// TIA Portal V18 export
// export: Created 2025-12-01T12:38:33.7594151Z, ExportSetting None, DisplayName Totally Integrated Automation Portal, DisplayVersion V18 Update 5, DisplayName TIA Portal Openness, DisplayVersion V18 Update 5, DisplayName TIA Portal Teamcenter Gateway, DisplayVersion V18, DisplayName TIA Portal Version Control Interface, DisplayVersion V18, DisplayName STEP 7 Professional, DisplayVersion V18 Update 5, DisplayName STEP 7 Safety, DisplayVersion V18, DisplayName WinCC Professional, DisplayVersion V18 Update 5
FUNCTION "ST10Cyl_interface41-50" : Void   // FC1024, LAD
{ S7_Optimized_Access := 'FALSE' }
// stored: AutoNumber false, SetENOAutomatically false
   VAR_INPUT
      AlwaysON : Bool;
      E_stop : Bool;
   END_VAR
   VAR_TEMP
      tTest : Bool;
   END_VAR
BEGIN

REGION Network 1 (SCL): Cylinder 41-50 IO Interface (SCL)
   //Cylinder41 IO  K-reserveLifting3LiftingCylinder
   //Input
   "ST10Cylinder".Cy[41].In.WorkPositionSensor := "iK-reserveLifting3LiftingCylinderInWP";
   "ST10Cylinder".Cy[41].In.HomePositionSensor := "iK-reserveLifting3LiftingCylinderInHP";
   //Output
   "oK-reserveLifting3LiftingCylinderToWP" := "ST10Cylinder".Cy[41].Out.GoWorkPosition;
   "oK-reserveLifting3LiftingCylinderToHP" := "ST10Cylinder".Cy[41].Out.GoHomePosition;

   //Cylinder42 IO  K-reserveLifting3PalletLocationCylinder
   //Input
   "ST10Cylinder".Cy[42].In.WorkPositionSensor := "iK-reserveLifting3PalletLocationCylinderInWP";
   "ST10Cylinder".Cy[42].In.HomePositionSensor := "iK-reserveLifting3PalletLocationCylinderInHP";
   //Output
   "oK-reserveLifting3PalletLocationCylinderToWP" := "ST10Cylinder".Cy[42].Out.GoWorkPosition;
   "oK-reserveLifting3PalletLocationCylinderToHP" := "ST10Cylinder".Cy[42].Out.GoHomePosition;

   //Cylinder43 IO  K-reserveLoadingStopperCylinder1
   //Input
   "ST10Cylinder".Cy[43].In.WorkPositionSensor := "oK-reserveLoadingStopperCylinder1_ToWP";
   "ST10Cylinder".Cy[43].In.HomePositionSensor := "oK-reserveLoadingStopperCylinder1_ToHP";
   //Output
   "oK-reserveLoadingStopperCylinder1_ToWP" := "ST10Cylinder".Cy[43].Out.GoWorkPosition;
   "oK-reserveLoadingStopperCylinder1_ToHP" := "ST10Cylinder".Cy[43].Out.GoHomePosition;

   //Cylinder44 IO  K-reserveLoadingStopperCylinder2
   //Input
   "ST10Cylinder".Cy[44].In.WorkPositionSensor := "oK-reserveLoadingStopperCylinder2_ToWP";
   "ST10Cylinder".Cy[44].In.HomePositionSensor := "oK-reserveLoadingStopperCylinder2_ToHP";
   //Output
   "oK-reserveLoadingStopperCylinder2_ToWP" := "ST10Cylinder".Cy[44].Out.GoWorkPosition;
   "oK-reserveLoadingStopperCylinder2_ToHP" := "ST10Cylinder".Cy[44].Out.GoHomePosition;

   //Cylinder45 IO  K-reserveLoadingStopperCylinder3
   //Input
   "ST10Cylinder".Cy[45].In.WorkPositionSensor := "oK-reserveLoadingStopperCylinder3_ToWP";
   "ST10Cylinder".Cy[45].In.HomePositionSensor := "oK-reserveLoadingStopperCylinder3_ToHP";
   //Output
   "oK-reserveLoadingStopperCylinder3_ToWP" := "ST10Cylinder".Cy[45].Out.GoWorkPosition;
   "oK-reserveLoadingStopperCylinder3_ToHP" := "ST10Cylinder".Cy[45].Out.GoHomePosition;

   //Cylinder46 K-reserveLoadingStopperCylinder4
   //Input
   "ST10Cylinder".Cy[46].In.WorkPositionSensor := "oK-reserveLoadingStopperCylinder4_ToWP";
   "ST10Cylinder".Cy[46].In.HomePositionSensor := "oK-reserveLoadingStopperCylinder4_ToHP";
   //Output
   "oK-reserveLoadingStopperCylinder4_ToWP" := "ST10Cylinder".Cy[46].Out.GoWorkPosition;
   "oK-reserveLoadingStopperCylinder4_ToHP" := "ST10Cylinder".Cy[46].Out.GoHomePosition;

   //Cylinder47 K-reserveTakeStopperCylinder1
   //Input
   "ST10Cylinder".Cy[47].In.WorkPositionSensor := "oK-reserveTakeStopperCylinder1_ToWP";
   "ST10Cylinder".Cy[47].In.HomePositionSensor := "oK-reserveTakeStopperCylinder1_ToHP";
   //Output
   "oK-reserveTakeStopperCylinder1_ToWP" := "ST10Cylinder".Cy[47].Out.GoWorkPosition;
   "oK-reserveTakeStopperCylinder1_ToHP" := "ST10Cylinder".Cy[47].Out.GoHomePosition;

   //Cylinder48 K-reserveTakeStopperCylinder2
   //Input
   "ST10Cylinder".Cy[48].In.WorkPositionSensor := "oK-reserveTakeStopperCylinder2_ToWP";
   "ST10Cylinder".Cy[48].In.HomePositionSensor := "oK-reserveTakeStopperCylinder2_ToHP";
   //Output
   "oK-reserveTakeStopperCylinder2_ToWP" := "ST10Cylinder".Cy[48].Out.GoWorkPosition;
   "oK-reserveTakeStopperCylinder2_ToHP" := "ST10Cylinder".Cy[48].Out.GoHomePosition;

   //Cylinder49 K-reserveTakeStopperCylinder3
   //Input
   "ST10Cylinder".Cy[49].In.WorkPositionSensor := "oK-reserveTakeStopperCylinder3_ToWP";
   "ST10Cylinder".Cy[49].In.HomePositionSensor := "oK-reserveTakeStopperCylinder3_ToHP";
   //Output
   "oK-reserveTakeStopperCylinder3_ToWP" := "ST10Cylinder".Cy[49].Out.GoWorkPosition;
   "oK-reserveTakeStopperCylinder3_ToHP" := "ST10Cylinder".Cy[49].Out.GoHomePosition;

   (*
   //Cylinder50 K-reserveLoadingStopperCylinder4_2
   // //Input
   "ST10Cylinder".Cy[50].In.WorkPositionSensor := "oK-reserveLoadingStopperCylinder4_2";
   "ST10Cylinder".Cy[50].In.HomePositionSensor := NOT "oK-reserveLoadingStopperCylinder4_2";
   // //Output
   "oK-reserveLoadingStopperCylinder4_2" := "ST10Cylinder".Cy[50].Out.GoWorkPosition;
   // "Feeding washer  lift Cylinder ToHP" := "ST10Cylinder".Cy[50].Out.GoHomePosition;
   *)
END_REGION

REGION Network 2: CY41 interface K-reserveLifting3LiftingCylinder
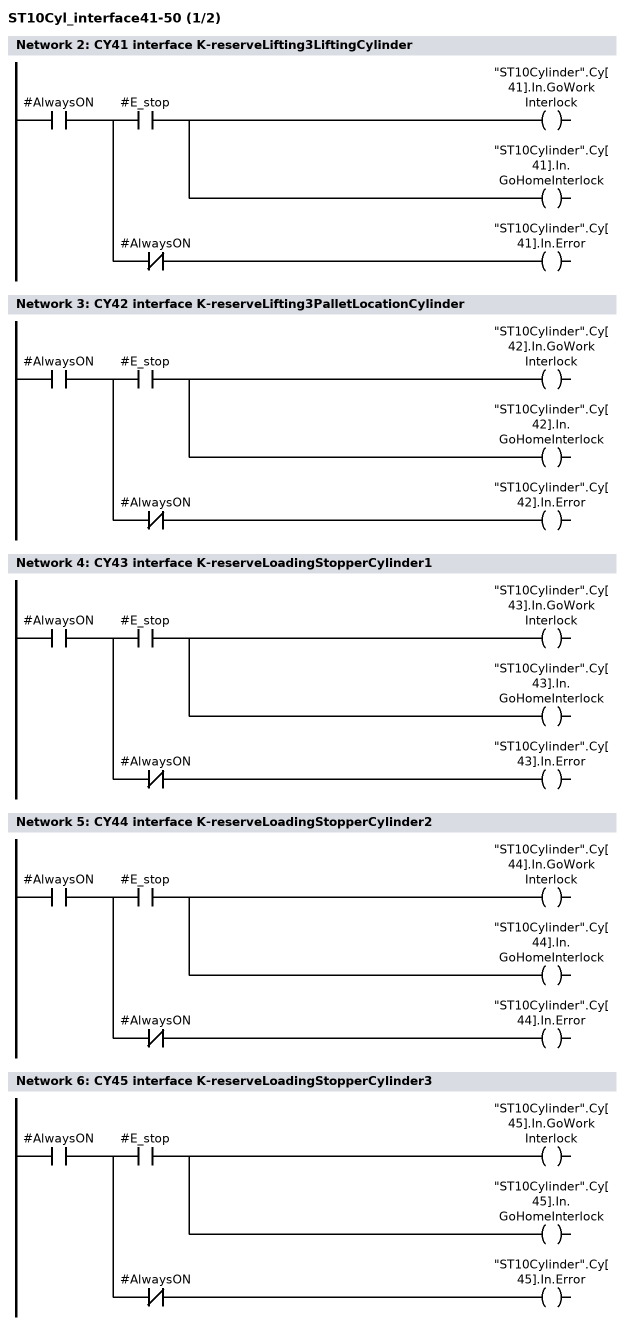
   RUNG wire#powerrail
      Contact( #AlwaysON )
      wire#w1
      Contact( #E_stop )
      wire#w2
      Coil( "ST10Cylinder".Cy[41].In.GoWorkInterlock )
   END_RUNG
   RUNG wire#w2
      Coil( "ST10Cylinder".Cy[41].In.GoHomeInterlock )
   END_RUNG
   RUNG wire#w1
      I_Contact( #AlwaysON )
      Coil( "ST10Cylinder".Cy[41].In.Error )
   END_RUNG
   // the same network as SCL:
   "ST10Cylinder".Cy[41].In.GoWorkInterlock := #AlwaysON AND #E_stop;
   "ST10Cylinder".Cy[41].In.GoHomeInterlock := #AlwaysON AND #E_stop;
   "ST10Cylinder".Cy[41].In.Error := #AlwaysON AND NOT #AlwaysON;
END_REGION

REGION Network 3: CY42 interface K-reserveLifting3PalletLocationCylinder
   RUNG wire#powerrail
      Contact( #AlwaysON )
      wire#w1
      Contact( #E_stop )
      wire#w2
      Coil( "ST10Cylinder".Cy[42].In.GoWorkInterlock )
   END_RUNG
   RUNG wire#w2
      Coil( "ST10Cylinder".Cy[42].In.GoHomeInterlock )
   END_RUNG
   RUNG wire#w1
      I_Contact( #AlwaysON )
      Coil( "ST10Cylinder".Cy[42].In.Error )
   END_RUNG
   // the same network as SCL:
   "ST10Cylinder".Cy[42].In.GoWorkInterlock := #AlwaysON AND #E_stop;
   "ST10Cylinder".Cy[42].In.GoHomeInterlock := #AlwaysON AND #E_stop;
   "ST10Cylinder".Cy[42].In.Error := #AlwaysON AND NOT #AlwaysON;
END_REGION

REGION Network 4: CY43 interface K-reserveLoadingStopperCylinder1
   RUNG wire#powerrail
      Contact( #AlwaysON )
      wire#w1
      Contact( #E_stop )
      wire#w2
      Coil( "ST10Cylinder".Cy[43].In.GoWorkInterlock )
   END_RUNG
   RUNG wire#w2
      Coil( "ST10Cylinder".Cy[43].In.GoHomeInterlock )
   END_RUNG
   RUNG wire#w1
      I_Contact( #AlwaysON )
      Coil( "ST10Cylinder".Cy[43].In.Error )
   END_RUNG
   // the same network as SCL:
   "ST10Cylinder".Cy[43].In.GoWorkInterlock := #AlwaysON AND #E_stop;
   "ST10Cylinder".Cy[43].In.GoHomeInterlock := #AlwaysON AND #E_stop;
   "ST10Cylinder".Cy[43].In.Error := #AlwaysON AND NOT #AlwaysON;
END_REGION

REGION Network 5: CY44 interface K-reserveLoadingStopperCylinder2
   RUNG wire#powerrail
      Contact( #AlwaysON )
      wire#w1
      Contact( #E_stop )
      wire#w2
      Coil( "ST10Cylinder".Cy[44].In.GoWorkInterlock )
   END_RUNG
   RUNG wire#w2
      Coil( "ST10Cylinder".Cy[44].In.GoHomeInterlock )
   END_RUNG
   RUNG wire#w1
      I_Contact( #AlwaysON )
      Coil( "ST10Cylinder".Cy[44].In.Error )
   END_RUNG
   // the same network as SCL:
   "ST10Cylinder".Cy[44].In.GoWorkInterlock := #AlwaysON AND #E_stop;
   "ST10Cylinder".Cy[44].In.GoHomeInterlock := #AlwaysON AND #E_stop;
   "ST10Cylinder".Cy[44].In.Error := #AlwaysON AND NOT #AlwaysON;
END_REGION

REGION Network 6: CY45 interface K-reserveLoadingStopperCylinder3
   RUNG wire#powerrail
      Contact( #AlwaysON )
      wire#w1
      Contact( #E_stop )
      wire#w2
      Coil( "ST10Cylinder".Cy[45].In.GoWorkInterlock )
   END_RUNG
   RUNG wire#w2
      Coil( "ST10Cylinder".Cy[45].In.GoHomeInterlock )
   END_RUNG
   RUNG wire#w1
      I_Contact( #AlwaysON )
      Coil( "ST10Cylinder".Cy[45].In.Error )
   END_RUNG
   // the same network as SCL:
   "ST10Cylinder".Cy[45].In.GoWorkInterlock := #AlwaysON AND #E_stop;
   "ST10Cylinder".Cy[45].In.GoHomeInterlock := #AlwaysON AND #E_stop;
   "ST10Cylinder".Cy[45].In.Error := #AlwaysON AND NOT #AlwaysON;
END_REGION

REGION Network 7: CY46 interface K-reserveLoadingStopperCylinder4
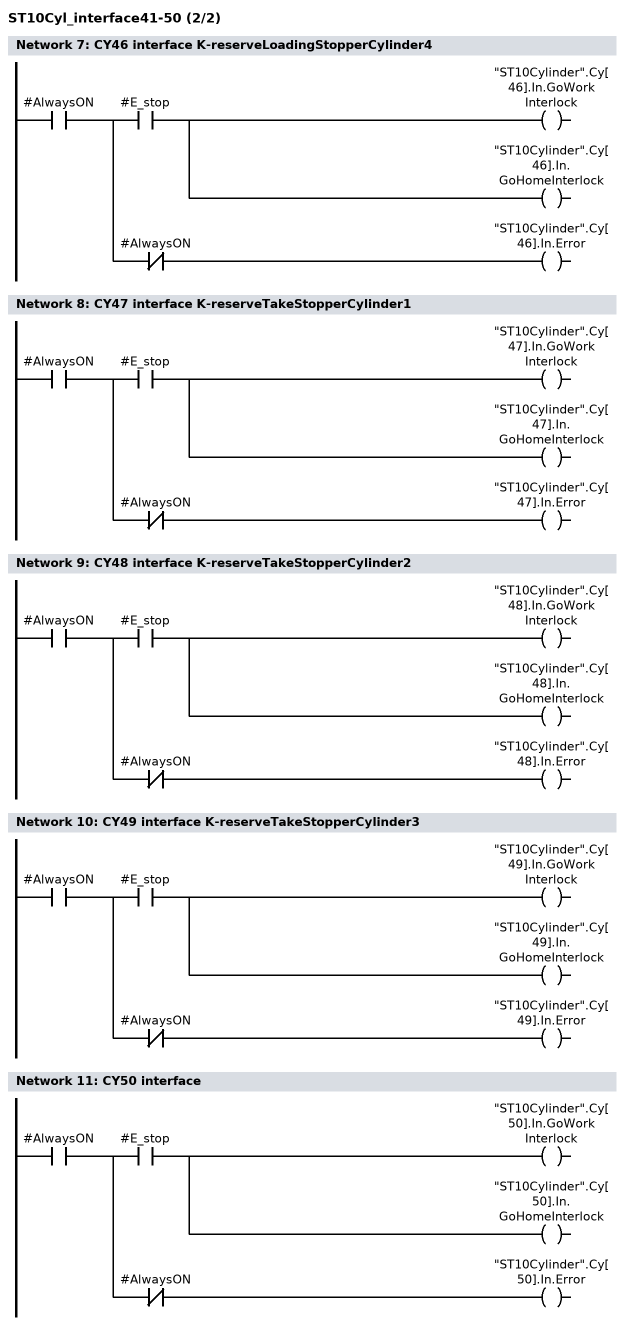
   RUNG wire#powerrail
      Contact( #AlwaysON )
      wire#w1
      Contact( #E_stop )
      wire#w2
      Coil( "ST10Cylinder".Cy[46].In.GoWorkInterlock )
   END_RUNG
   RUNG wire#w2
      Coil( "ST10Cylinder".Cy[46].In.GoHomeInterlock )
   END_RUNG
   RUNG wire#w1
      I_Contact( #AlwaysON )
      Coil( "ST10Cylinder".Cy[46].In.Error )
   END_RUNG
   // the same network as SCL:
   "ST10Cylinder".Cy[46].In.GoWorkInterlock := #AlwaysON AND #E_stop;
   "ST10Cylinder".Cy[46].In.GoHomeInterlock := #AlwaysON AND #E_stop;
   "ST10Cylinder".Cy[46].In.Error := #AlwaysON AND NOT #AlwaysON;
END_REGION

REGION Network 8: CY47 interface K-reserveTakeStopperCylinder1
   RUNG wire#powerrail
      Contact( #AlwaysON )
      wire#w1
      Contact( #E_stop )
      wire#w2
      Coil( "ST10Cylinder".Cy[47].In.GoWorkInterlock )
   END_RUNG
   RUNG wire#w2
      Coil( "ST10Cylinder".Cy[47].In.GoHomeInterlock )
   END_RUNG
   RUNG wire#w1
      I_Contact( #AlwaysON )
      Coil( "ST10Cylinder".Cy[47].In.Error )
   END_RUNG
   // the same network as SCL:
   "ST10Cylinder".Cy[47].In.GoWorkInterlock := #AlwaysON AND #E_stop;
   "ST10Cylinder".Cy[47].In.GoHomeInterlock := #AlwaysON AND #E_stop;
   "ST10Cylinder".Cy[47].In.Error := #AlwaysON AND NOT #AlwaysON;
END_REGION

REGION Network 9: CY48 interface K-reserveTakeStopperCylinder2
   RUNG wire#powerrail
      Contact( #AlwaysON )
      wire#w1
      Contact( #E_stop )
      wire#w2
      Coil( "ST10Cylinder".Cy[48].In.GoWorkInterlock )
   END_RUNG
   RUNG wire#w2
      Coil( "ST10Cylinder".Cy[48].In.GoHomeInterlock )
   END_RUNG
   RUNG wire#w1
      I_Contact( #AlwaysON )
      Coil( "ST10Cylinder".Cy[48].In.Error )
   END_RUNG
   // the same network as SCL:
   "ST10Cylinder".Cy[48].In.GoWorkInterlock := #AlwaysON AND #E_stop;
   "ST10Cylinder".Cy[48].In.GoHomeInterlock := #AlwaysON AND #E_stop;
   "ST10Cylinder".Cy[48].In.Error := #AlwaysON AND NOT #AlwaysON;
END_REGION

REGION Network 10: CY49 interface K-reserveTakeStopperCylinder3
   RUNG wire#powerrail
      Contact( #AlwaysON )
      wire#w1
      Contact( #E_stop )
      wire#w2
      Coil( "ST10Cylinder".Cy[49].In.GoWorkInterlock )
   END_RUNG
   RUNG wire#w2
      Coil( "ST10Cylinder".Cy[49].In.GoHomeInterlock )
   END_RUNG
   RUNG wire#w1
      I_Contact( #AlwaysON )
      Coil( "ST10Cylinder".Cy[49].In.Error )
   END_RUNG
   // the same network as SCL:
   "ST10Cylinder".Cy[49].In.GoWorkInterlock := #AlwaysON AND #E_stop;
   "ST10Cylinder".Cy[49].In.GoHomeInterlock := #AlwaysON AND #E_stop;
   "ST10Cylinder".Cy[49].In.Error := #AlwaysON AND NOT #AlwaysON;
END_REGION

REGION Network 11: CY50 interface
   RUNG wire#powerrail
      Contact( #AlwaysON )
      wire#w1
      Contact( #E_stop )
      wire#w2
      Coil( "ST10Cylinder".Cy[50].In.GoWorkInterlock )
   END_RUNG
   RUNG wire#w2
      Coil( "ST10Cylinder".Cy[50].In.GoHomeInterlock )
   END_RUNG
   RUNG wire#w1
      I_Contact( #AlwaysON )
      Coil( "ST10Cylinder".Cy[50].In.Error )
   END_RUNG
   // the same network as SCL:
   "ST10Cylinder".Cy[50].In.GoWorkInterlock := #AlwaysON AND #E_stop;
   "ST10Cylinder".Cy[50].In.GoHomeInterlock := #AlwaysON AND #E_stop;
   "ST10Cylinder".Cy[50].In.Error := #AlwaysON AND NOT #AlwaysON;
END_REGION
END_FUNCTION
